SUBAPPLICATION PAGE_1 (* Subapplication Type *)
  (* Standard: 61499-2 *)
  (* Version 1.0, 2023-02-07, franz *)
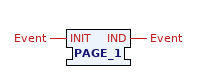
  EVENT_INPUT
    INIT;
  END_EVENT
  EVENT_OUTPUT
    IND;
  END_EVENT
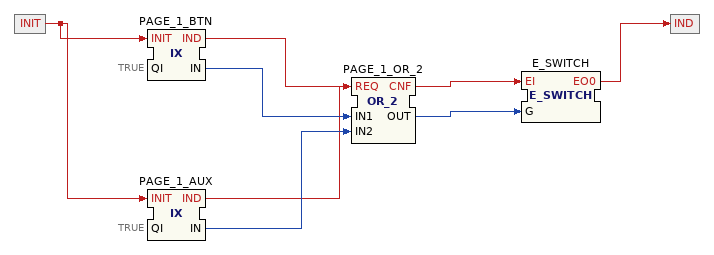
  FBS
    PAGE_1_BTN : IX(QI := TRUE);
    PAGE_1_AUX : IX(QI := TRUE);
    PAGE_1_OR_2 : OR_2;
    E_SWITCH : E_SWITCH;
  END_FBS
  EVENT_CONNECTIONS
    INIT TO PAGE_1_BTN.INIT;
    INIT TO PAGE_1_AUX.INIT;
    PAGE_1_BTN.IND TO PAGE_1_OR_2.REQ;
    PAGE_1_AUX.IND TO PAGE_1_OR_2.REQ;
    PAGE_1_OR_2.CNF TO E_SWITCH.EI;
    E_SWITCH.EO0 TO IND;
  END_CONNECTIONS
  DATA_CONNECTIONS
    PAGE_1_BTN.IN TO PAGE_1_OR_2.IN1;
    PAGE_1_AUX.IN TO PAGE_1_OR_2.IN2;
    PAGE_1_OR_2.OUT TO E_SWITCH.G;
  END_CONNECTIONS
END_SUBAPPLICATION
